// TIA Portal V20 export
// export: Created 2025-12-01T14:57:19.0319631Z, ExportSetting None, DisplayName Totally Integrated Automation Portal, DisplayVersion V20 Update 3, DisplayName TIA Portal Openness, DisplayVersion V20 Update 3, DisplayName TIA Portal Version Control Interface, DisplayVersion V20 Update 3, DisplayName STEP 7 Professional, DisplayVersion V20 Update 3, DisplayName STEP 7 Safety, DisplayVersion V20 Update 2, DisplayName WinCC Basic/Comfort/Advanced, DisplayVersion V20 Update 3, DisplayName WinCC Professional, DisplayVersion V20 Update 3, DisplayName WinCC Unified, DisplayVersion V20 Update 3
DATA_BLOCK "DB221_FIFO_ORDENES_S3"   // DB221
{ S7_Optimized_Access := 'FALSE' }
AUTHOR : ROUTER
NAME : 20130623
VERSION : 3.1
// stored: AutoNumber false
   VAR
      FIFO : Array[0.."CTE_MaxMesas"] of Struct   // 0 a 50 scanners y 1 ordenes posibles en la FIFO
         Posicion { S7_SetPoint := 'True'} : Array[1..5] of "ROUT_Orden_Fifo_Scanner";
      END_STRUCT;
   END_VAR
BEGIN
END_DATA_BLOCK
